(* IEC 61131-3 sources: myCodes/Stone/07.02.2022 - OOPs Approach/MPx_One_New/Mpx_One_Source_Code/MPx_One/3. USHPXMPX010A1/USHPXMPX010A1/MPXone_Medium/Widgets, 6 files *)

(* ---- Wizard.st ---- *)
USING System.UI;
USING HEOneRow;
USING System.Math;
USING System;
USING System.Globalization;
USING Libs.CustomGas;

VAR_GLOBAL
    tmpWiz: WizParams;

    tmpConfOk : ARRAY[0..NUM_WIZ_PARAMS] OF BOOL;
    wizCanEnd : BOOL := FALSE;
END_VAR

VAR_GLOBAL CONSTANT
    {IF NOT DEF(MPXONE_ADVANCED)}
    NUM_WIZ_PARAMS : USINT := 12;
    {ELSE}
    NUM_WIZ_PARAMS : USINT := 13;
    {ENDIF}
END_VAR

TYPE
    WizData : UNION
        bool : BOOL;
        usint : USINT;
        sint : SINT;
        real : REAL;
    END_UNION;

    WizStruct: STRUCT
        (** Master or slave configuration *)
        In : WizData := (bool := FALSE);
        (** Number or slave devices *)
        Sn : WizData := (usint := 0);
        (** Number or slave devices *)
        H0 : WizData := (usint := 199);
        (** BMS protocol selection *)
        H3 : WizData := (bool := TRUE);
        (** Type of probes on Group1 (S1, S2 and S3) *)
        _P1 : WizData := (bool := TRUE);
        (** Valve type *)
        {IF NOT DEF(MPXONE_ADVANCED)}
        P1 :  WizData := (usint := 0);
        {ELSE}
        P1 :  WizData := (usint := 1); //valve present by default in PMXone Advanced
        {ENDIF}
        (** Refrigerant type *)
        PH :  WizData := (usint := 3);
        (** Type of probes on Group2 (S4 and S5) *)
        _P2 :  WizData := (usint := 2);
        (** Type of probes on Group3 (S6)*)
        _P3 :  WizData := (usint := 1);
        (** Channel of suction temperature probe *)
        _FD :  WizData := (usint := 0);
        (** Channel of evaporation pressure probe *)
        _FE :  WizData := (usint := 0);
        (** Maximum of evaporation pressure probe *)
        _UE :  WizData := (real := 9.3);
        (** Minimum of evaporation pressure probe *)
        _LE :  WizData := (real := -1.0);
         {IF DEF(MPXONE_ADVANCED)}
        (** Type of probes on Group3 (S8)*)
        _P5 :  WizData := (usint := 1);
        {ENDIF}
    END_STRUCT;

    WizParams : UNION
        Fct : WizStruct;
        Arr : ARRAY [0..NUM_WIZ_PARAMS] OF WizData;    // Biggest data type
    END_UNION;

END_TYPE

{METADATA DEFAULT_SELECTABLE "TRUE"}
{METADATA WIDGET_TYPE "Text"}
{METADATA PREVIEW_STRING "Wiz"}
{METADATA SUPPORT_TERMINALS "SevenSegments;HEOneRow"}
CLASS WizardWidget

	VAR PUBLIC
		x,y : INT;	//auto-assigned
        Acronim : STRING[3];
        ValIndex : USINT := 0;
	END_VAR

	VAR PRIVATE
        (*not modify, just for widget*)
        StringWrite : STRING[5];

        showValue : BOOL;

        tmpVal : WizData;

        isReal : BOOL;
        isBool : BOOL;
        isUsint : BOOL;
        isSint : BOOL;

        Min, Max : REAL;

        _UOM : UOM := UOM#NONE;
	END_VAR

	METHOD PUBLIC Init
        // Reset the visualization
        //ValIndex := 0;
        showValue := FALSE;

        // Get value of Wiz parameter
        tmpVal :=  tmpWiz.Arr[ValIndex];

        // Get type of Wiz parameter
        CASE ValIndex OF
            0, 3 , 4: THIS.isBool := TRUE;
            1, 2, 5..8: THIS.isUsint := TRUE;
            9..10: THIS.isSint := TRUE;
            11..12: THIS.isReal := TRUE;
            13: THIS.isSint := TRUE;
            _UOM := UOM#BAR;
        END_CASE;

        // Get limits
        CASE ValIndex OF
            1: THIS.Min := 0.0; THIS.Max := 9.0; // parameter Sn
            2: THIS.Min := 1.0; THIS.Max := 247.0; // parameter H0
            5: THIS.Min := 0.0; THIS.Max := 6.0; // parameter P1
            6: THIS.Min := 0; THIS.Max := 40; // parameter PH
            7: THIS.Min := 1; THIS.Max := 3; // parameter /P2
            8: THIS.Min := 0; THIS.Max := 4; // parameter /P3
            {IF NOT DEF (MPXONE_ADVANCED)}
                9: THIS.Min := -4; THIS.Max := 6; // parameter /Fd
                10: THIS.Min := -4; THIS.Max := 6; // parameter /FE
            {ENDIF}
            {IF DEF (MPXONE_ADVANCED)}
                9: THIS.Min := -4; THIS.Max := 8; // parameter /Fd
                10: THIS.Min := -4; THIS.Max := 8; // parameter /FE
            {ENDIF}
            11: THIS.Min := EvapMin; THIS.Max := 200.0; // parameter /UE
            12: THIS.Min := -1.0; THIS.Max := EvapMax; // parameter /LE

            {IF DEF (MPXONE_ADVANCED)}
            13: THIS.Min := 1; THIS.Max := 2; // parameter /P5
            {ENDIF}
        END_CASE;

	END_METHOD

	METHOD PUBLIC Draw

        IF showValue THEN
            IF THIS.isBool THEN
                StringWrite := TO_STRING(TO_USINT(tmpVal.bool));
            ELSIF THIS.isUsint THEN
                StringWrite := TO_STRING(tmpVal.usint);
            ELSIF THIS.isSint THEN
                StringWrite := TO_STRING(tmpVal.sint);
            ELSIF THIS.isReal THEN
                StringWrite := REAL_TO_DISPLAY(tmpVal.real);
            END_IF;
        ELSE
            StringWrite := Acronim;
        END_IF;

        (*draw the string*)
        DrawString(StringWrite, 0, 0);

    END_METHOD

	{METADATA ACTION "KEY_DOWN"}
	METHOD PUBLIC KeyDown
        IF showValue THEN
            IF THIS.isBool THEN
                tmpVal.bool := NOT tmpVal.bool;

            ELSIF THIS.isUsint THEN
                tmpVal.usint := tmpVal.usint - 1;

                IF tmpVal.usint > TO_USINT(THIS.Max) THEN
                    tmpVal.usint := TO_USINT(THIS.Max);
                END_IF;

                IF tmpVal.usint < TO_USINT(THIS.Min) THEN
                    tmpVal.usint := TO_USINT(THIS.Max);
                END_IF;
            ELSIF THIS.isSint THEN
                tmpVal.sint := tmpVal.sint - 1;

                IF tmpVal.sint < TO_SINT(THIS.Min) THEN
                    tmpVal.sint := TO_SINT(THIS.Max);
                END_IF;
            ELSIF THIS.isReal THEN
                tmpVal.real := tmpVal.real - 0.1;

                IF tmpVal.real < THIS.Min THEN
                    tmpVal.real := THIS.Max;
                END_IF;
            END_IF;
        ELSE
            GoToNextMask();
        END_IF;
	END_METHOD

    {METADATA ACTION "KEY_UP"}
 	METHOD PUBLIC KeyUp
        IF showValue THEN
            IF THIS.isBool THEN
                tmpVal.bool := NOT tmpVal.bool;

            ELSIF THIS.isUsint THEN
                tmpVal.usint := tmpVal.usint + 1;

                IF tmpVal.usint > TO_USINT(THIS.Max) THEN
                    tmpVal.usint := TO_USINT(THIS.Min);
                END_IF;
            ELSIF THIS.isSint THEN
                tmpVal.sint := tmpVal.sint + 1;

                IF tmpVal.sint > TO_SINT(THIS.Max) THEN
                    tmpVal.sint := TO_SINT(THIS.Min);
                END_IF;
            ELSIF THIS.isReal THEN
                tmpVal.real := tmpVal.real + 0.1;

                IF tmpVal.real > THIS.Max THEN
                    tmpVal.real := THIS.Min;
                END_IF;
            END_IF;
        ELSE
            GoToPreviousMask();
        END_IF;
    END_METHOD

    {METADATA ACTION "KEY_PRG"}
 	METHOD PUBLIC KeyPrg
        VAR
            i : INT;
        END_VAR

        showValue := NOT showValue;

        IF NOT showValue THEN
            tmpConfOk[ValIndex] := TRUE;
            tmpWiz.Arr[ValIndex] := tmpVal;

            // Check if wizard can finish
            wizCanEnd := TRUE;
            FOR i := TO_INT(LOWER_BOUND(tmpWiz.Arr, 1)) TO TO_INT(UPPER_BOUND(tmpWiz.Arr, 1)) DO
                IF i = 1 AND NOT tmpWiz.Fct.In.bool THEN CONTINUE; END_IF;
                IF i = 4 OR i = 5 AND isBasic THEN CONTINUE; END_IF;
                IF i > 5 AND NOT VlvPresent THEN CONTINUE; END_IF;

                wizCanEnd := wizCanEnd AND tmpConfOk[i];
            END_FOR;
        END_IF;
    END_METHOD

    {METADATA ACTION "KEY_ALARM"}
 	METHOD PUBLIC KeyAlarm
        //showValue := FALSE;

        // blockHmi := TRUE;
        // IdxVis := 1;
        // LedOnArrow := FALSE;
        // GoToMask(MaskList#mMain);
        // Navigation := FALSE;
    END_METHOD

END_CLASS

(* ---- WidgetMain.st ---- *)
USING System.UI;
USING HEOneRow;
USING System.Math;
USING System;
USING System.Timer;
USING System.Globalization;
USING System.io;

VAR_GLOBAL
            // same of Ain_offset but orderd by channel (introduced for compatibility)
    U_offset    : ARRAY[1..LIB_IO_MAX_U_CH] OF REAL;
END_VAR

{METADATA DEFAULT_SELECTABLE "FALSE"}
{METADATA WIDGET_TYPE "Text"}
{METADATA PREVIEW_STRING "VAL"}
{METADATA SUPPORT_TERMINALS "SevenSegments;HEOneRow"}
CLASS MainWidget

	VAR PUBLIC
		x,y : INT;	//auto-assigned
	END_VAR

	VAR PRIVATE
        (*not modify, just for widget*)
        StringVal_HMImain_TMP : STRING[5];
        StringVal_HMIrem_TMP : STRING[5];
        StringAlrm : STRING[4];
        i, startI : INT := 1;
        TON_CAROSEL : TON;
        ShowStringAlarm : BOOL;
        ShowStringOff : BOOL;
        ShowStringDef : BOOL;
        FoundAlrm : BOOL;

        DefRT : R_TRIG;
        DefStoredT : STRING[5];
        DefStoredT_RemHMI : STRING[5];
        keepHMIDef : BOOL;
        DefStoredTVal : REAL;
        HMIVisValue : REAL;
	END_VAR

	METHOD PUBLIC Init

	END_METHOD

    METHOD PRIVATE ValueToStr : STRING[5]
        VAR_INPUT
            uomVal : UOM;
            realVal : REAL;
        END_VAR
        VAR
            _INT : INT;
            _REAL : REAL;
        END_VAR

        CONVERT_UOM_ZONE(realVal, uomVal, _REAL, GetUIZone());

        _INT := TO_INT(TRUNC(_REAL));
        IF DisDecPointMainVar THEN
            ValueToStr := TO_STRING(_INT);
        ELSE
            ValueToStr := REAL_TO_DISPLAY(_REAL);
        END_IF;

    END_METHOD

    METHOD PRIVATE ValueToStr : STRING[5]
        VAR_INPUT
            realVal : REAL;
        END_VAR
        VAR
            _INT : INT;
        END_VAR

        _INT := TO_INT(TRUNC(realVal));
        IF DisDecPointMainVar THEN
            ValueToStr := TO_STRING(_INT);
        ELSE
            ValueToStr := REAL_TO_DISPLAY(realVal);
        END_IF;

    END_METHOD

    METHOD PRIVATE showErrToDisp : BOOL
        VAR_INPUT
            HMI_Sel : USINT;
        END_VAR

        CASE HMI_Sel OF
            1..8: // Physical probes
                showErrToDisp := Alarms.Al.Al_PrbBroken[HMI_Sel].Info.Active;

            9: // Control probe
                showErrToDisp := DutySettings;

            10: // Virtual probe
                showErrToDisp := VirtualComposition = 0 AND AirOffBroken OR VirtualComposition = 100 AND AirOnBroken;

            11..14: // Serial probes
                IF HMI_Sel - 10 < 1 THEN
                    showErrToDisp := TRUE;
                ELSE
                    showErrToDisp := Alarms.Al.Al_SerialInputs[HMI_Sel - 10].Info.Active;
                END_IF;
            ELSE
                showErrToDisp := FALSE;
        END_CASE;
    END_METHOD

    METHOD PRIVATE createStringToDisp : STRING[5]
        VAR_INPUT
            HMI_Sel : USINT;
        END_VAR

        VAR
            PhysPrb_tmp : REAL;
            CtlPrb_tmp : REAL;
            VirtPrb_tmp : REAL;
        END_VAR

        Offset_Fct2Ch();
        CASE HMI_Sel OF
            0: // Terminal disabled
                createStringToDisp := '';
                HMIVisValue := 0.0;

            1..8: // Physical probes
                PhysPrb_tmp := TO_REAL(Libs.Math.Round((U[HMI_Sel].r + U_offset[HMI_Sel]) * 10.0)) / 10.0;
                createStringToDisp := ValueToStr(PhysPrb_tmp);
                HMIVisValue := PhysPrb_tmp;

            9: // Control probe
                CtlPrb_tmp := TO_REAL(Libs.Math.Round(RegProbe * 10.0)) / 10.0;
                createStringToDisp := ValueToStr(UOM_OF(RegProbe), CtlPrb_tmp);
                HMIVisValue := CtlPrb_tmp;

            10: // Virtual probe
                VirtPrb_tmp := TO_REAL(Libs.Math.Round(VirtualProbe * 10.0)) / 10.0;
                createStringToDisp := ValueToStr(UOM_OF(VirtualProbe), VirtPrb_tmp);
                HMIVisValue := VirtPrb_tmp;

            11..14: // Serial probes (without offset)
                createStringToDisp := ValueToStr(SerialInputs[HMI_Sel - 10].r);
                HMIVisValue := SerialInputs[HMI_Sel - 10].r;

            15: // Temperature setpoint
                createStringToDisp := ValueToStr(UOM_OF(TempSetP), TempSetP);
                HMIVisValue := TempSetP;

            {IF NOT DEF(MPXONE_BASIC)}
            16: //Actual superheat reading
                IF (Ain_Cfg.Arr[4].Ch > 0 AND Ain_Cfg.Arr[5].Ch > 0) OR (ValveCnf = 6) THEN
                    createStringToDisp := ValueToStr(UOM_OF(ActualSH), ActualSH);
                    HMIVisValue := ActualSH;
                ELSE
                    createStringToDisp := '----';
                    HMIVisValue := 0.0;
                END_IF;

            {ENDIF}
            ELSE
                createStringToDisp := '';
                HMIVisValue := 0.0;
        END_CASE;

    END_METHOD

	METHOD PUBLIC Draw
        VAR
            showErr_HMImain : BOOL;
            showErr_HMIrem : BOOL;
        END_VAR

        (*draw the string*)
        {REGION MAIN_VALUE_TO_SHOW}
        (*choose what is shown in the main mask*)
        (*value is replicated in two versions:
         -REAL(with decimal point)
        -UINT(without decimal point)*)

        // Remote HMI
        StringVal_HMIrem_TMP := createStringToDisp(HmiRemSel);
        showErr_HMIrem := showErrToDisp(HmiRemSel);
        IF showErr_HMIrem THEN
            StringVal_HMIrem_TMP := TO_STRING(999);
        END_IF;

        // Main HMI
        StringVal_HMImain_TMP := createStringToDisp(HmiMainSel);
        showErr_HMImain := showErrToDisp(HmiMainSel);
        IF showErr_HMImain THEN
            StringVal_HMImain_TMP := TO_STRING(999);
        END_IF;

        // Show version during startup
        IF firstCycle THEN
            StringVal_HMImain_TMP := 'r' + TO_STRING(__PROJ_VER_MAJOR__) + '.' + TO_STRING(__PROJ_VER_MINOR__);
            StringVal_HMIrem_TMP := StringVal_HMImain_TMP;
        END_IF;

        // Text during defrost
        DefRT(CLK := (DfrStatus > DFR_IDLE) OR DfrNatural);
        IF DefRT.Q THEN
            DefStoredT_RemHMI := StringVal_HMIrem_TMP;
            DefStoredT := StringVal_HMImain_TMP;

        //TRAC #95
        // save last value shown to manage the visualization of the main value to show
        // after the end of the defrost if "d6" = 1 or 2
            IF NOT(keepHMIDef) THEN

                Offset_Fct2Ch();
                 CASE HmiMainSel OF
                    0: // Terminal disabled
                        DefStoredTVal := 0.0;

                    1..8: // Physical probes
                        DefStoredTVal := TO_REAL(Libs.Math.Round((U[HMIMainSel].r) + U_offset[HMIMainSel] * 10.0)) / 10.0;

                    9: // Control probe
                        DefStoredTVal := TO_REAL(Libs.Math.Round(RegProbe * 10.0)) / 10.0;

                    10: // Virtual probe
                        DefStoredTVal := TO_REAL(Libs.Math.Round(VirtualProbe * 10.0)) / 10.0;

                    11..14: // Serial probes (without offset)
                       DefStoredTVal := SerialInputs[HMIMainSel - 10].r;

                    15: // Temperature setpoint
                        DefStoredTVal := TempSetP;

                    {IF NOT DEF(MPXONE_BASIC)}
                    16: //Actual superheat reading
                        IF (Ain_Cfg.Arr[4].Ch > 0 AND Ain_Cfg.Arr[5].Ch > 0) OR (ValveCnf = 6) THEN
                            DefStoredTVal := ActualSH;
                        ELSE
                            DefStoredTVal := 0.0;
                        END_IF;

                    {ENDIF}
                    ELSE
                        DefStoredTVal := 0.0;
                END_CASE;
            END_IF;

        END_IF;

        ShowStringDef := FALSE;
        IF DfrStatus > DFR_IDLE OR DfrNatural THEN
            CASE HmiMainDef OF
                0:
                    StringVal_HMImain_TMP := DefStoredT;
                    StringVal_HMIrem_TMP := DefStoredT_RemHMI;
                    ShowStringDef := TRUE;
                    keepHMIDef := FALSE;

                1:
                    StringVal_HMImain_TMP := DefStoredT;
                    StringVal_HMIrem_TMP := DefStoredT_RemHMI;
                    keepHMIDef := TRUE;

                2:
                    StringVal_HMImain_TMP := 'DEF';
                    StringVal_HMIrem_TMP :=  'DEF';
                    keepHMIDef := TRUE;
            END_CASE;

        //TRAC #95
        ELSIF keepHMIDef THEN //if HMIMainDef (d6) =1 or 2 after the defrost keep showing the last temperature before the start of the defrost

                StringVal_HMImain_TMP := DefStoredT;
                StringVal_HMIrem_TMP := DefStoredT_RemHMI;

            // stop showing the
            IF (RegProbe<=ActualTempSetpoint OR (TempDiff2>0 AND RegProbe<= ActualTemp2Setpoint) OR NOT(UnitOn) OR HMIVisValue<=DefStoredTVal OR DfrHiBypassEnd) THEN
                keepHMIDef := FALSE;
            END_IF;

        END_IF;

        {ENDREGION }

        ActCarosel := ActCarosel OR NOT UnitOn OR ShowStringDef;
        TON_CAROSEL(IN := ActCarosel,PT := t#3s);
        IF TON_CAROSEL.Q AND NOT firstCycle THEN
            TON_CAROSEL(IN := FALSE,PT := t#0s);

            FoundAlrm := FALSE;
            startI := i;
            WHILE NOT FoundAlrm AND NOT ShowStringAlarm DO
                IF ActiveAlm[i] > 0 AND Alarms.Arr[i].StrCode <> '' THEN

                    StringAlrm := Alarms.Arr[i].StrCode;
                    FoundAlrm := TRUE;
                END_IF;
                i := i + 1;
                IF i > TO_INT(UPPER_BOUND(ActiveAlm,1)) THEN
                    i := TO_INT(LOWER_BOUND(ActiveAlm,1));
                END_IF;

                // Prevent never ending loop
                IF i = startI THEN
                    IF NOT FoundAlrm THEN
                        ActCarosel := FALSE; //TRAC #117 - reset carousel if no alarms are anymore present
                    END_IF;

                    EXIT;
                END_IF;

            END_WHILE;

            IF NOT UnitOn THEN
                ShowStringAlarm := (NOT ShowStringAlarm XOR ShowStringOff) AND FoundAlrm;
                ShowStringOff := NOT ShowStringOff XOR ShowStringAlarm;
            ELSE
                ShowStringAlarm := NOT ShowStringAlarm;
                ShowStringOff := FALSE;
            END_IF;

        END_IF;

        IF ShowStringAlarm AND ActCarosel THEN
            IF ShowStringDef THEN
                DrawString('DEF', 0, 0);
            ELSE
                DrawString(StringAlrm, 0, 0);
            END_IF;
            {IF NOT DEF(NO_MPXONE_REPEATER)}
            IF RemoteHMIAlrms THEN
                IF ShowStringDef THEN
                    mpxRepeater.SetText(1, 'DEF');
                ELSE
                    mpxRepeater.SetText(1, StringAlrm);
                END_IF;
            END_IF;
            {ENDIF}
        ELSIF ShowStringOff  AND ActCarosel THEN
            DrawString('OFF', 0, 0);
            {IF NOT DEF(NO_MPXONE_REPEATER)}
            IF RemoteHMIAlrms THEN
                mpxRepeater.SetText(1, 'OFF');
            END_IF;
            {ENDIF}
        ELSE
            DrawString(StringVal_HMImain_TMP , 0, 0);

            {IF NOT DEF(NO_MPXONE_REPEATER)}
            mpxRepeater.SetText(1, StringVal_HMIrem_TMP);
            {ENDIF}
        END_IF;
    END_METHOD

END_CLASS

(**Populate U_offset array with offset present in Ain_Offset*)
FUNCTION Offset_Fct2Ch
    VAR
        i   : DINT;
    END_VAR

            //populate U_Offset used for channel I/O oriented logic (Vs Fct orinted)
            // (serial probe have no ofset)
    FOR i := 1 TO UPPER_BOUND(Ain_Offset.Arr,1) DO
        IF Ain_Cfg.Arr[i].Ch > 0 THEN
            U_offset[Ain_Cfg.Arr[i].Ch] := Ain_Offset.Arr[i];
        END_IF;
    END_FOR;

END_FUNCTION

(* ---- Default.st ---- *)
USING System.UI;
USING HEOneRow;
USING System.Timer;
USING System;

{METADATA DEFAULT_SELECTABLE "FALSE"}
{METADATA WIDGET_TYPE "Text"}
{METADATA PREVIEW_STRING "DEF"}
{METADATA SUPPORT_TERMINALS "SevenSegments;HEOneRow"}
CLASS DefaultWidget

	VAR PUBLIC
		x,y : INT;	//auto-assigned
	END_VAR

	VAR PRIVATE
        value : USINT;
        CnfRes : BOOL := TRUE;
        errTON : TON;
	END_VAR

	METHOD PUBLIC Init
        // Reset the visualization
        value := 0;
	END_METHOD

	METHOD PUBLIC Draw

        (*draw the string*)
        DrawString(TO_STRING(value), 0, 0);

        errTON(IN := NOT CnfRes, PT := T#5s);
        CnfRes := CnfRes OR errTON.Q;

        SetBuzzer(NOT CnfRes);
        LEDAlmOn := NOT CnfRes;

    END_METHOD

	{METADATA ACTION "KEY_DOWN"}
	METHOD PUBLIC KeyDown
        value := value - 1;
        // Unsigned lower bound check
        IF value > 2 THEN
            value := 2;
        END_IF;
	END_METHOD

    {METADATA ACTION "KEY_UP"}
 	METHOD PUBLIC KeyUp
        value := value + 1;
        // Unsigned upper bound check
        IF value > 2 THEN
            value := 0;
        END_IF;
    END_METHOD

    {METADATA ACTION "KEY_PRG"}
 	METHOD PUBLIC KeyPrg

        // Wait until PRG is released
        IF BlockHmi THEN
            RETURN;
        END_IF;

        CASE value OF
            0: // Reset carel default
            ResCarelSets := TRUE;
            THIS.Close(MaskList#WIZ_In);

            1: // MT Configuration
            CnfRes := SetConfiguration('C1');
            IF CnfRes THEN
                //GoToMask(MaskList#mMain);
                THIS.Close(MaskList#mMain);
                StartupReset := FALSE;
            END_IF;

            2: // LT Configuration
            CnfRes := SetConfiguration('C2');
            IF CnfRes THEN
                //GoToMask(MaskList#mMain);
                THIS.Close(MaskList#mMain);
                StartupReset := FALSE;
            END_IF;

        END_CASE;

    END_METHOD

    METHOD Close
        VAR_INPUT
            msk : MaskList;
        END_VAR

        //StartupReset := FALSE;
        LedBlinkArrow := FALSE;
        //WizDone := FALSE;

        GoToMask(msk);

    END_METHOD

    {METADATA ACTION "KEY_PROGRAM_RELEASE"}
    METHOD PUBLIC DefaultPROGRAM_RELEASE

        IF BlockHmi THEN
           BlockHmi := FALSE;
        END_IF;

    END_METHOD

END_CLASS

(* ---- ReadOnly.st ---- *)
USING System.UI;
USING HEOneRow;
USING System.Math;
USING System;
USING System.Globalization;

{METADATA DEFAULT_SELECTABLE "FALSE"}
{METADATA WIDGET_TYPE "Text"}
{METADATA PREVIEW_STRING "R/O"}
{METADATA SUPPORT_TERMINALS "SevenSegments;HEOneRow"}
CLASS ReadOnlyWidget

	VAR PUBLIC
		x,y : INT;	//auto-assigned
        Acronim : STRING[3];
        ValIndex : USINT := 1;
	END_VAR

	VAR PRIVATE
        (*not modify, just for widget*)
        StringWrite : STRING[5];

        showValue : BOOL;

	END_VAR

	METHOD PUBLIC Init
        // Reset the visualization
        //ValIndex := 0;
        THIS.showValue := FALSE;
	END_METHOD

	METHOD PUBLIC Draw
        VAR
            _UOM : UOM;
            _REAL : REAL;
        END_VAR

        _UOM := UOM#NONE;
        // Mostly Celsius
        IF ValIndex >= 1 AND ValIndex <= 13 THEN
            _UOM := UOM#CELSIUS;
        END_IF;
        CASE ValIndex OF
            5:  _UOM := UOM#BAR;
            10: _UOM := UOM#PERCENT_rH;
            14: _UOM := UOM#CELSIUS;
            16: _UOM := UOM#PERCENT;
        END_CASE;

        CONVERT_UOM_ZONE(RegValues[ValIndex], _UOM, _REAL, GetUIZone());

        IF THIS.showValue THEN
            StringWrite := REAL_TO_DISPLAY(_REAL);
        ELSE
            StringWrite := Acronim;
        END_IF;

        (*draw the string*)
        DrawString(StringWrite, 0, 0);

    END_METHOD

	{METADATA ACTION "KEY_DOWN"}
	METHOD PUBLIC KeyDown
        THIS.showValue := FALSE;
        GoToNextMask();
	END_METHOD

    {METADATA ACTION "KEY_UP"}
 	METHOD PUBLIC KeyUp
        THIS.showValue := FALSE;
        GoToPreviousMask();
    END_METHOD

    {METADATA ACTION "KEY_PRG"}
 	METHOD PUBLIC KeyPrg
        THIS.showValue := NOT THIS.showValue;
    END_METHOD

    {METADATA ACTION "KEY_PROGRAM_RELEASE"}
    METHOD PUBLIC KeyProgramRelease

    END_METHOD

    {METADATA ACTION "KEY_ALARM"}
 	METHOD PUBLIC KeyAlarm
        THIS.showValue := FALSE;

        // blockHmi := TRUE;
        // IdxVis := 1;
        // LedOnArrow := FALSE;
        // GoToMask(MaskList#mMain);
        // Navigation := FALSE;
    END_METHOD

END_CLASS

(* ---- WidgetAlarm.st ---- *)
USING System.UI;
USING HEOneRow;
USING System.Math;
USING System;

    (*
        +--------------------------------+            /|
        |                                |           /  ------ -  -
        | Insert WIDGET source code here |          |
        |                                |           \  ------ -  -
        +--------------------------------+            \|
    *)

{REGION Alarm}

    {METADATA DEFAULT_SELECTABLE "FALSE"}
    {METADATA WIDGET_TYPE "Text"}
    {METADATA PREVIEW_STRING "ALM"}
    {METADATA SUPPORT_TERMINALS "SevenSegments;HEOneRow"}
    CLASS AlarmWidget

    	VAR PUBLIC
    		x,y : INT;	//auto-assigned
    	END_VAR

    	VAR PRIVATE
            (*not modify, just for widget*)
            StringWrite : STRING[3];
            //CompactAlrmAct : ARRAY[1..NUM_ALARMS] OF UINT;
            CompactAlrmAct : ARRAY[1..NUM_ALARMS + NUM_WARN_STATUS] OF UINT;
            i : INT := 1;
            k : INT := 1;
            IdxVis : INT := 1;

    	END_VAR

    	METHOD PUBLIC Init

    	END_METHOD

    	METHOD PUBLIC Draw
        (*draw the string*)
        (*mantain ready alway the first element*)
        LedOnArrow := TRUE;
        k := TO_INT(LOWER_BOUND(CompactAlrmAct,1));
        FOR i := TO_INT(LOWER_BOUND(ActiveAlm,1)) TO TO_INT(UPPER_BOUND(ActiveAlm,1)) DO
            (*clear the list before to write*)
            CompactAlrmAct[i] := 0;
            (*compact the list of active alarm*)
            IF ActiveAlm[i] > 0 THEN
                CompactAlrmAct[k] := TO_UINT(i);
                //CompactAlrmAct[k] := ActiveAlm[i];
                k := k + 1;
            END_IF;
        END_FOR;

        IF IdxVis = k OR IdxVis = TO_INT(LOWER_BOUND(CompactAlrmAct,1)) THEN
            StringWrite := 'ESC';
        END_IF;
        (*last index, go to first*)
        IF IdxVis >= k OR IdxVis < TO_INT(LOWER_BOUND(CompactAlrmAct,1)) THEN
            IF IdxVis < TO_INT(LOWER_BOUND(CompactAlrmAct,1)) THEN
                IdxVis := k;
            END_IF;

            IF IdxVis > k THEN
                IdxVis := TO_INT(LOWER_BOUND(CompactAlrmAct,1));
            END_IF;

        ELSE
            (*reset compact*)
            k := TO_INT(LOWER_BOUND(CompactAlrmAct,1));
            IF CompactAlrmAct[TO_INT(LOWER_BOUND(CompactAlrmAct,1))] = 0 THEN
                (*write no alarm*)
                StringWrite := ' NO';
            ELSE
                (*write determinated alarm*)
                StringWrite := Alarms.Arr[CompactAlrmAct[IdxVis]].StrCode;
                //StringWrite := ALARM_CODES[CompactAlrmAct[IdxVis]];
            END_IF;
        END_IF;

        DrawString(StringWrite, 0, 0);

        END_METHOD

    	{METADATA ACTION "KEY_DOWN"}
    	METHOD PUBLIC KeyDown
            IdxVis := IdxVis + 1;
    	END_METHOD

        {METADATA ACTION "KEY_UP"}
     	METHOD PUBLIC KeyUp
            IdxVis := IdxVis - 1;
        END_METHOD

        {METADATA ACTION "KEY_PRG"}
     	METHOD PUBLIC KeyPrg

            IF StringWrite = 'ESC' THEN
                blockHmi := TRUE;
                IdxVis := TO_INT(LOWER_BOUND(CompactAlrmAct,1));
                LedOnArrow := FALSE;
                GoToMask(MaskList#mMain);
                Navigation := FALSE;
            END_IF;
        END_METHOD

        {METADATA ACTION "KEY_ALARM"}
     	METHOD PUBLIC KeyAlarm
            blockHmi := TRUE;
            IdxVis := TO_INT(LOWER_BOUND(CompactAlrmAct,1));
            LedOnArrow := FALSE;
            GoToMask(MaskList#mMain);
            Navigation := FALSE;
        END_METHOD

    END_CLASS

{ENDREGION }

(* ---- WidgetAlarmsHyst.st ---- *)
USING System.UI;
USING HEOneRow;
USING System.Math;
USING System.Timer;
USING System;
USING System.Alarm;

    (*
        +--------------------------------+            /|
        |                                |           /  ------ -  -
        | Insert WIDGET source code here |          |
        |                                |           \  ------ -  -
        +--------------------------------+            \|
    *)

{REGION Alarm_Hyst}

    {METADATA DEFAULT_SELECTABLE "FALSE"}
    {METADATA WIDGET_TYPE "Text"}
    {METADATA PREVIEW_STRING "ALM"}
    {METADATA SUPPORT_TERMINALS "SevenSegments;HEOneRow"}
    CLASS AlarmHystWidget

    	VAR PUBLIC
    		x,y : INT;	//auto-assigned
    	END_VAR

    	VAR PRIVATE
            (*not modify, just for widget*)
            StringWrite : STRING[3];
            CompactAlrmHyst : ARRAY[1..NUM_ALARMS_HYST] OF ArrayCompactAlrmHyst;
    	END_VAR

    	METHOD PUBLIC Init

    	END_METHOD

    	METHOD PUBLIC Draw

            (*draw the string*)
            (*mantain ready alway the first element*)
            LedOnArrow := TRUE;

            THIS.createAlrmCodeArray();

            CASE AlrmHyst_idx OF
                ALRMHYST_ENUM#CODE:
                        StringWrite := CompactAlrmHyst[IdxVis_AlrmHyst].Code_Str;

                ALRMHYST_ENUM#YEAR:
                    IF CompactAlrmHyst[IdxVis_AlrmHyst].Year > 2000 THEN
                        StringWrite := TO_STRING(CompactAlrmHyst[IdxVis_AlrmHyst].Year - 2000);
                    ELSE
                        StringWrite := STRING_ALM_HYST_EMPTY;
                    END_IF;
                ALRMHYST_ENUM#MONTH:
                    StringWrite := TO_STRING(CompactAlrmHyst[IdxVis_AlrmHyst].Month);
                ALRMHYST_ENUM#DAY:
                    StringWrite := TO_STRING(CompactAlrmHyst[IdxVis_AlrmHyst].Day);
                ALRMHYST_ENUM#HOUR:
                    StringWrite := TO_STRING(CompactAlrmHyst[IdxVis_AlrmHyst].Hour);
                ALRMHYST_ENUM#MIN:
                    StringWrite := TO_STRING(CompactAlrmHyst[IdxVis_AlrmHyst].Minute);
                ALRMHYST_ENUM#DURATION:
                    StringWrite := TO_STRING(CompactAlrmHyst[IdxVis_AlrmHyst].Duration);
                ALRMHYST_ENUM#WRITE_ESC:
                    StringWrite := 'ESC';
            END_CASE;

            IF StringWrite <> STRING_ALM_HYST_EMPTY THEN
                DrawString(StringWrite, 0, 0);
            ELSE
                DrawString(StringWrite, 0, 1);
            END_IF;
        END_METHOD

    	{METADATA ACTION "KEY_DOWN"}
    	METHOD PUBLIC KeyDown
            IF StringWrite = STRING_ALM_HYST_EMPTY THEN
                AlrmHyst_idx := ALRMHYST_ENUM#WRITE_ESC;
            ELSIF AlrmHyst_idx = ALRMHYST_ENUM#WRITE_ESC  THEN
                AlrmHyst_idx := ALRMHYST_ENUM#CODE;
            ELSE
                AlrmHyst_idx := AlrmHyst_idx + 1;
            END_IF;
    	END_METHOD

        {METADATA ACTION "KEY_UP"}
     	METHOD PUBLIC KeyUp
            IF StringWrite = STRING_ALM_HYST_EMPTY THEN
                AlrmHyst_idx := ALRMHYST_ENUM#WRITE_ESC;
            ELSIF AlrmHyst_idx = ALRMHYST_ENUM#CODE  THEN
                AlrmHyst_idx := ALRMHYST_ENUM#WRITE_ESC;
            ELSE
                AlrmHyst_idx := AlrmHyst_idx - 1;
            END_IF;
        END_METHOD

        {METADATA ACTION "KEY_PRG"}
     	METHOD PUBLIC KeyPrg

        END_METHOD

        {METADATA ACTION "KEY_PROGRAM_RELEASE"}
        METHOD PUBLIC KeyPrgRelease
            IF StringWrite = 'ESC' THEN
                blockHmi := TRUE;
                IdxVis_AlrmHyst := 0;
                LedOnArrow := TRUE;
                PopLastMask();
                AlrmHyst_idx := ALRMHYST_ENUM#CODE;
                Navigation := FALSE;
            END_IF;
        END_METHOD

        {METADATA ACTION "KEY_ALARM"}
     	METHOD PUBLIC KeyAlarm
            blockHmi := TRUE;
            IdxVis_AlrmHyst := 0;
            LedOnArrow := FALSE;
            GoToMask(MaskList#mMain);
            Navigation := FALSE;
        END_METHOD

        METHOD PRIVATE createAlrmCodeArray
            VAR
                i : INT;
//                k : INT := 1;
                memIdx : INT := 1;
                Al_Year : UINT;
                Al_Month : UINT;
                Al_Day : UINT;
                Al_Hour : UINT;
                AL_Minute : UINT;
                AL_Second : UINT;
                Al_Millisecond : UINT;
                timeStampStop, timeStampStart : DATE_AND_TIME;
            END_VAR

            FOR i := 1 TO TO_INT(UPPER_BOUND(THIS.CompactAlrmHyst,1)) DO
                THIS.CompactAlrmHyst[i].Code_Str := '---';
                THIS.CompactAlrmHyst[i].Year := 0;
                THIS.CompactAlrmHyst[i].Month := 0;
                THIS.CompactAlrmHyst[i].Day := 0;
                THIS.CompactAlrmHyst[i].Hour := 0;
                THIS.CompactAlrmHyst[i].Minute := 0;
                THIS.CompactAlrmHyst[i].Duration := 0;
            END_FOR;

            memIdx := 1;
            FOR i := 1 TO TO_INT(UPPER_BOUND(LogAlarms,1)) DO
                IF LogAlarms[i].Code <> 0 AND LogAlarms[i].Status = 0 THEN
                    THIS.CompactAlrmHyst[memIdx].Code_Str := findAlrmCodeStr(LogAlarms[i].Code);
                    timeStampStart := LogAlarms[i].TimeStamp;
                    SPLIT_DT(timeStampStart, Al_Year, Al_Month, Al_Day, Al_Hour, AL_Minute, AL_Second, Al_Millisecond);
                    THIS.CompactAlrmHyst[memIdx].Year := Al_Year;
                    THIS.CompactAlrmHyst[memIdx].Month := Al_Month;
                    THIS.CompactAlrmHyst[memIdx].Day := Al_Day;
                    THIS.CompactAlrmHyst[memIdx].Hour := Al_Hour;
                    THIS.CompactAlrmHyst[memIdx].Minute := AL_Minute;
                    timeStampStop := findLogAlrmTimeStamp(LogAlarms[i].Code, AlarmStatus#Stop, i);
                    THIS.CompactAlrmHyst[memIdx].Duration := TO_UDINT(timeStampStop - timeStampStart) / 60000;
                    IF THIS.CompactAlrmHyst[memIdx].Duration > 999 THEN
                        THIS.CompactAlrmHyst[memIdx].Duration := 999;
                    END_IF;

                    memIdx := memIdx + 1;
                    IF memIdx > TO_INT(UPPER_BOUND(CompactAlrmHyst,1)) THEN
                        memIdx := 1;
                    END_IF;
                END_IF;
            END_FOR;

        END_METHOD

        METHOD PRIVATE findAlrmCodeStr : STRING[3]
            VAR_INPUT
                Al_Code_tmp : UINT;
            END_VAR

            IF Al_Code_tmp <= TO_UINT(UPPER_BOUND(Alarms.Arr,1)) THEN
                findAlrmCodeStr := Alarms.Arr[AL_Code_tmp].StrCode;
            ELSE
                findAlrmCodeStr := '---';
            END_IF;
        END_METHOD

        METHOD PRIVATE findLogAlrmTimeStamp : DATE_AND_TIME
            VAR_INPUT
                Al_code_tmp : UINT;
                startStop_type : AlarmStatus;
                startIndx : INT;
            END_VAR

            VAR
                i : INT;
            END_VAR

            startIndx := startIndx + 1;
            FOR i := startIndx TO TO_INT(UPPER_BOUND(LogAlarms,1)) DO
                IF LogAlarms[i].Code = Al_Code_tmp AND LogAlarms[i].Status >= startStop_type THEN
                    findLogAlrmTimeStamp := LogAlarms[i].TimeStamp;
                    EXIT;
                END_IF;
            END_FOR;

        END_METHOD

    END_CLASS
{ENDREGION }
